DATA_BLOCK "DB_KeyenceCheckerIV3"
{ S7_Optimized_Access := 'TRUE' }
VERSION : 0.1
NON_RETAIN
// ATTRIBUTES
// AUTO_NUMBER = False
// BLOCK_NUMBER = 2101
// END_ATTRIBUTES
   VAR
      aDev : Array[1..4] of "ST_KeyenceCheckerIV3";
   END_VAR


BEGIN
   aDev[1].Para.nInAdr1 := 465;
   aDev[1].Para.nInAdr2 := 466;
   aDev[1].Para.nInAdr3 := 467;
   aDev[1].Para.nInAdr4 := 468;
   aDev[1].Para.nInAdr5 := 354;
   aDev[1].Para.nInAdr6 := 469;
   aDev[1].Para.nInAdr7 := 470;
   aDev[1].Para.nInAdr8 := 471;
   aDev[1].Para.nInAdr9 := 472;
   aDev[1].Para.nInAdr10 := 473;
   aDev[1].Para.nInAdr11 := 474;
   aDev[1].Para.nInAdr12 := 475;
   aDev[1].Para.nInAdr13 := 476;
   aDev[1].Para.nInAdr14 := 477;
   aDev[1].Para.nInAdr15 := 478;
   aDev[1].Para.nInAdr16 := 479;
   aDev[1].Para.nInAdr17 := 480;
   aDev[1].Para.nInAdr18 := 481;
   aDev[1].Para.nInAdr19 := 482;
   aDev[1].Para.nInAdr20 := 483;
   aDev[1].Para.nInAdr21 := 484;
   aDev[1].Para.nInAdr22 := 485;
   aDev[1].Para.nInAdr23 := 486;
   aDev[1].Para.nInAdr24 := 487;
   aDev[1].Para.nInAdr25 := 488;
   aDev[1].Para.nInAdr26 := 489;
   aDev[1].Para.nInAdr27 := 509;
   aDev[1].Para.nInAdr28 := 510;
   aDev[1].Para.nInAdr29 := 511;
   aDev[1].Para.nInAdr30 := 512;
   aDev[1].Para.nInAdr31 := 513;
   aDev[1].Para.nInAdr32 := 514;
   aDev[1].Para.nInAdr33 := 515;
   aDev[1].Para.nInAdr34 := 516;
   aDev[1].Para.nInAdr35 := 517;
   aDev[1].Para.nInAdr36 := 518;
   aDev[1].Para.nInAdr37 := 519;
   aDev[1].Para.nInAdr38 := 520;
   aDev[1].Para.nInAdr39 := 521;
   aDev[1].Para.nInAdr40 := 522;
   aDev[1].Para.nInAdr41 := 523;
   aDev[1].Para.nInAdr42 := 524;
   aDev[1].Para.nInAdr43 := 525;
   aDev[1].Para.nInAdr44 := 526;
   aDev[1].Para.nInAdr45 := 527;
   aDev[1].Para.nInAdr46 := 528;
   aDev[1].Para.nInAdr47 := 529;
   aDev[1].Para.nInAdr48 := 530;
   aDev[1].Para.nInAdr49 := 531;
   aDev[1].Para.nInAdr50 := 532;
   aDev[1].Para.nInAdr51 := 533;
   aDev[1].Para.nInAdr52 := 534;
   aDev[1].Para.nInAdr53 := 535;
   aDev[1].Para.nInAdr54 := 536;
   aDev[1].Para.nInAdr55 := 373;
   aDev[1].Para.nInAdr56 := 537;
   aDev[1].Para.nInAdr57 := 377;
   aDev[1].Para.nInAdr58 := 538;
   aDev[1].Para.nInAdr59 := 539;
   aDev[1].Para.nInAdr60 := 540;
   aDev[1].Para.nInAdr61 := 541;
   aDev[1].Para.nInAdr62 := 542;
   aDev[1].Para.nInAdr63 := 543;
   aDev[1].Para.nInAdr64 := 544;
   aDev[1].Para.nInAdr65 := 545;
   aDev[1].Para.nInAdr66 := 546;
   aDev[1].Para.nInAdr67 := 547;
   aDev[1].Para.nInAdr68 := 548;
   aDev[1].Para.nInAdr69 := 549;
   aDev[1].Para.nInAdr70 := 550;
   aDev[1].Para.nOutAdr1 := 464;
   aDev[2].Para.nInAdr1 := 435;
   aDev[2].Para.nInAdr2 := 434;
   aDev[2].Para.nInAdr3 := 433;
   aDev[2].Para.nInAdr4 := 432;
   aDev[2].Para.nInAdr5 := 431;
   aDev[2].Para.nInAdr6 := 430;
   aDev[2].Para.nInAdr7 := 429;
   aDev[2].Para.nInAdr8 := 428;
   aDev[2].Para.nInAdr9 := 427;
   aDev[2].Para.nInAdr10 := 426;
   aDev[2].Para.nInAdr11 := 425;
   aDev[2].Para.nInAdr12 := 424;
   aDev[2].Para.nInAdr13 := 423;
   aDev[2].Para.nInAdr14 := 422;
   aDev[2].Para.nInAdr15 := 421;
   aDev[2].Para.nInAdr16 := 420;
   aDev[2].Para.nInAdr17 := 419;
   aDev[2].Para.nInAdr18 := 418;
   aDev[2].Para.nInAdr19 := 417;
   aDev[2].Para.nInAdr20 := 416;
   aDev[2].Para.nInAdr21 := 415;
   aDev[2].Para.nInAdr22 := 414;
   aDev[2].Para.nInAdr23 := 413;
   aDev[2].Para.nInAdr24 := 412;
   aDev[2].Para.nInAdr25 := 411;
   aDev[2].Para.nInAdr26 := 410;
   aDev[2].Para.nInAdr27 := 409;
   aDev[2].Para.nInAdr28 := 408;
   aDev[2].Para.nInAdr29 := 407;
   aDev[2].Para.nInAdr30 := 406;
   aDev[2].Para.nInAdr31 := 405;
   aDev[2].Para.nInAdr32 := 404;
   aDev[2].Para.nInAdr33 := 403;
   aDev[2].Para.nInAdr34 := 402;
   aDev[2].Para.nInAdr35 := 401;
   aDev[2].Para.nInAdr36 := 400;
   aDev[2].Para.nInAdr37 := 399;
   aDev[2].Para.nInAdr38 := 398;
   aDev[2].Para.nInAdr39 := 397;
   aDev[2].Para.nInAdr40 := 396;
   aDev[2].Para.nInAdr41 := 395;
   aDev[2].Para.nInAdr42 := 394;
   aDev[2].Para.nInAdr43 := 393;
   aDev[2].Para.nInAdr44 := 392;
   aDev[2].Para.nInAdr45 := 391;
   aDev[2].Para.nInAdr46 := 390;
   aDev[2].Para.nInAdr47 := 389;
   aDev[2].Para.nInAdr48 := 388;
   aDev[2].Para.nInAdr49 := 387;
   aDev[2].Para.nInAdr50 := 386;
   aDev[2].Para.nInAdr51 := 385;
   aDev[2].Para.nInAdr52 := 384;
   aDev[2].Para.nInAdr53 := 383;
   aDev[2].Para.nInAdr54 := 382;
   aDev[2].Para.nInAdr55 := 381;
   aDev[2].Para.nInAdr56 := 380;
   aDev[2].Para.nInAdr57 := 379;
   aDev[2].Para.nInAdr58 := 376;
   aDev[2].Para.nInAdr59 := 375;
   aDev[2].Para.nInAdr60 := 374;
   aDev[2].Para.nInAdr61 := 372;
   aDev[2].Para.nInAdr62 := 371;
   aDev[2].Para.nInAdr63 := 370;
   aDev[2].Para.nInAdr64 := 369;
   aDev[2].Para.nInAdr65 := 368;
   aDev[2].Para.nInAdr66 := 367;
   aDev[2].Para.nInAdr67 := 366;
   aDev[2].Para.nInAdr68 := 365;
   aDev[2].Para.nInAdr69 := 364;
   aDev[2].Para.nInAdr70 := 363;
   aDev[2].Para.nOutAdr1 := 436;

END_DATA_BLOCK

